PROGRAM WaterBath_Control
VAR
	
	Estop_Temp : bool;

END_VAR

IF GVL_Waterbath.Waterbath_StopwithSystem THEN		//if the pelletizer estop is pressed AND the setting for system stop is set, then stop with an estop.
	Estop_Temp := GVL_Pelletizer.MyPelletizer.Pelletizer_STO;
ELSE
	Estop_Temp := TRUE;
END_IF




IF GVL_Waterbath.Waterbath_StartwithSystem THEN
	GVL_Waterbath.Waterbath_Start := GVL_Pelletizer.MyPelletizer.Pelletizer_Start;
END_IF




IF GVL_Waterbath.Waterbath_Start AND Estop_Temp THEN
	GVL_Waterbath.Pump_Start := TRUE;
ELSE
	GVL_Waterbath.Pump_Start := FALSE;
END_IF


GVL_Waterbath.Waterbath_Local_Control := NOT GVL_Waterbath.Waterbath_System_Control;

END_PROGRAM

(* stored: Version 1.1.0.1, ProductVersion 3.1.4024.12
   POU WaterBath_Control: Id {c7a292ea-ddf7-4656-b0aa-3864839d40cf}, SpecialFunc None *)
